{attribute 'TcGenerated'}
{attribute 'no-analysis'}
{attribute 'linkalways'}
// This function has been automatically generated from the project information.
VAR_GLOBAL CONSTANT
	{attribute 'const_non_replaced'}
	stLibVersion_TcUnit : ST_LibVersion := (iMajor := 2026, iMinor := 7, iBuild := 17, iRevision := 1, nFlags := 0, sVersion := '2026.7.17.1');
END_VAR

(* stored: Version 1.1.0.1
   GVL Global_Version: Id {899e68fc-21fd-4d89-beb5-fc369f4dda74} *)
